ABB RobotStudio station: palletizing.rspag

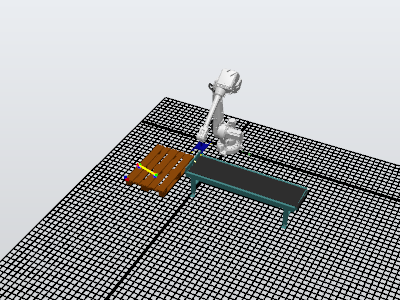
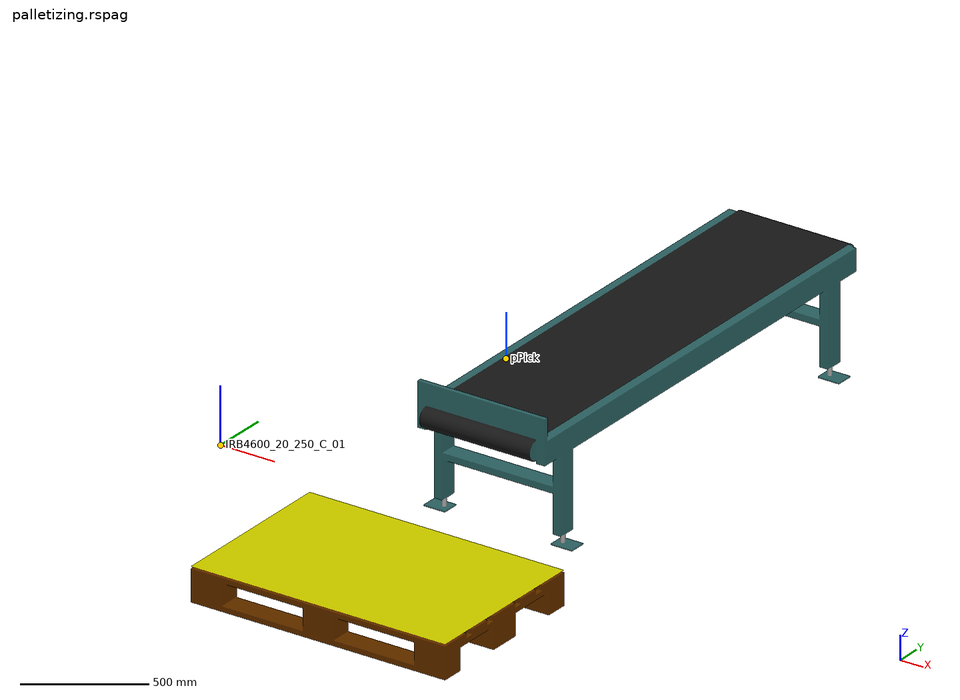
[picture v1: parts stored in the station drawn from their meshes, with robot base, taught points and paths (robot models come from the ABB library and are not in the file)]
--- station ---
Station palletizing (saved by RobotStudio 24.3.10958.1)
Controller IRB4600
  mechanical unit ROB_1: IRB4600_20_250_C_01, 6 joints, base frame (0, 0, 0) mm
Layout (positions relative to the parent item):
  - IRB4600_20_250_C_01 [mechanism, from %ABB.RobotStudio.Models.IRB4600%\IRB4600_20_250_C_G_01.rslib] at (0, 0, 0) mm; joint values [0.0538, -0.0275, 0.5427, 0, 1.0556, -1.517] (rad or m)
  - Belt Conveyor [part], size 703.5 x 2188.6 x 501 mm
  - Box [part], size 500 x 300 x 200 mm
  - SC_InFeeder [smart component]
      signals: DO doBoxInPos
      connections:
        LineSensor.SensorOut -> SC_InFeeder.doBoxInPos
        LineSensor.SensorOut -> LogicGate_2.InputA
        LogicGate_2.Output -> Source.Execute
    - Source [smart component, from Components\Source.rslib]
        properties: Source=Box; Copy=(none); Parent=(none); Position=[0 0 0]; Orientation=[0 0 0]; Transient=true; PhysicsBehavior=3
    - LineSensor [smart component, from Components\LineSensor.rslib]
        properties: Start=[1.3 -0.09 0.547]; End=[1.3 -0.03 0.547]; Radius=0; SensedPart=(none); SensedPoint=[1.3 -0.0800001220703125 0.547]; Length=0.06; Tag=(none)
      - _sensorPart_ [part], size 0 x 60 x 0 mm
    - LogicGate_2 [smart component, from Components\LogicGate.rslib]
        properties: Operator=NOT; Delay=0
  - Belt [part], size 529.1 x 2200.3 x 102.1 mm
  - Stop [part], size 600 x 20 x 100 mm
  - SC_VacuumTool [smart component] at (1300.02, 70, 1050.64) mm, rotated rx 180 ry 0 rz -90 deg
      signals: DI diAttach, DO doAttached
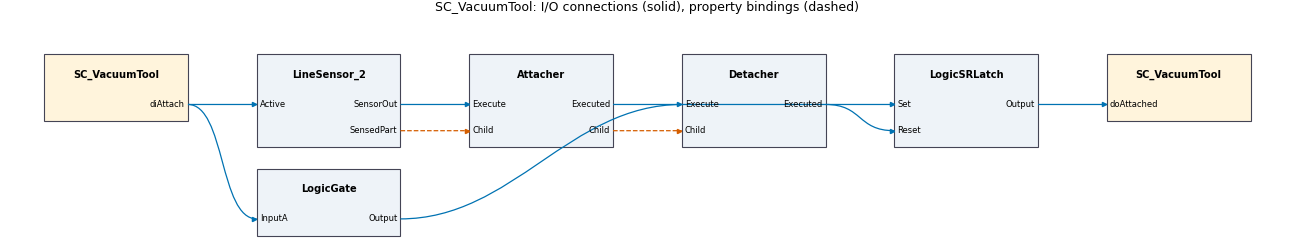
      connections:
        SC_VacuumTool.diAttach -> LineSensor_2.Active
        LineSensor_2.SensorOut -> Attacher.Execute
        Attacher.Executed -> LogicSRLatch.Set
        SC_VacuumTool.diAttach -> LogicGate.InputA
        LogicGate.Output -> Detacher.Execute
        Detacher.Executed -> LogicSRLatch.Reset
        LogicSRLatch.Output -> SC_VacuumTool.doAttached
        LineSensor_2.SensedPart => Attacher.Child
        Attacher.Child => Detacher.Child
    - LineSensor_2 [smart component, from Components\LineSensor.rslib]
        properties: Start=[0 0 0.1122]; End=[0 0 0.16]; Radius=0; SensedPart=(none); SensedPoint=[1.65000061035156 -1.05000048828125 0.345319213867188]; Length=0.0478; Tag=(none)
      - _sensorPart_ [part], size 0 x 0 x 47.8 mm
    - Attacher [smart component, from Components\Attacher.rslib]
        properties: Parent=Vacuum Tool; Flange=0; Child=(none); Mount=false; Offset=[0 0 0]; Orientation=[0 0 0]
    - Detacher [smart component, from Components\Detacher.rslib]
        properties: Child=(none); KeepPosition=true
    - LogicGate [smart component, from Components\LogicGate.rslib]
        properties: Operator=NOT; Delay=0
    - LogicSRLatch [smart component, from Components\LogicSRLatch.rslib]
    - Vacuum Tool [mechanism] at (0, 0, 0) mm
        TCP tVacuum at (0, 0, 150) mm
        links: Vacuum Tool
  - SC_OutFeeder [smart component]
      connections:
        PlaneSensor.SensorOut -> LogicGate.InputA
        LogicGate.Output -> Sink.Execute
        PlaneSensor.SensedPart => Sink.Object
    - EPAL Euro pallet [part] at (1900, -1200, 0) mm, rotated rx 0 ry 0 rz 90 deg, size 804.4 x 1206.6 x 151.6 mm
    - PlaneSensor [smart component, from Components\PlaneSensor.rslib]
        properties: Origin=[0.7 -1.2 0.154]; Axis1=[1.2 0 0]; Axis2=[0 0.8 0]; SensedPart=(none); Tag=(none)
      - _sensorPart_ [part], size 1200 x 800 x 0 mm
    - Sink [smart component, from Components\Sink.rslib]
        properties: Object=(none)
    - LogicGate [smart component, from Components\LogicGate.rslib]
        properties: Operator=NOP; Delay=2
Attachment: SC_VacuumTool is attached to IRB4600_20_250_C_01 / Link6
Station logic (signal -> signal, property => property):
  SC_VacuumTool.doAttached -> IRB4600.diVacuum
  IRB4600.doVacuum -> SC_VacuumTool.diAttach
  SC_InFeeder.doBoxInPos -> IRB4600.diBoxInPos
Targets, tools, work objects and paths stored in the station and not in the controller backup, written as RAPID:
! task T_ROB1
MODULE Module1
  PROC PickPart()
    MoveL pPick,v300,fine,tVacuum\WObj:=wobjInFeeder;
  ENDPROC
  PROC DropPart()
    MoveL Target_10,v300,fine,tVacuum\WObj:=wobjPallet;
    MoveL Target_20,v300,fine,tVacuum\WObj:=wobjPallet;
  ENDPROC
ENDMODULE


--- Backups/IRB4600/RAPID/TASK1/PROGMOD/CalibData.mod ---
MODULE CalibData
	PERS tooldata tVacuum:=[TRUE,[[0,0,150],[1,0,0,0]],[9,[0,0,100],[1,0,0,0],0,0,0]];
	TASK PERS wobjdata wobjInFeeder:=[FALSE,TRUE,"",[[0,0,0],[1,0,0,0]],[[1000,-80,497],[1,0,0,0]]];
    TASK PERS wobjdata wobjPallet:=[FALSE,TRUE,"",[[1900,-1200,144],[0.707106781,0,0,0.707106781]],[[0,0,0],[1,0,0,0]]];
ENDMODULE

--- Backups/IRB4600/RAPID/TASK1/PROGMOD/Module1.mod ---
MODULE Module1
    CONST robtarget pPick:=[[300.023,150,209.481],[0,-0.707106781,0.707106781,0],[0,0,0,0],[9E+09,9E+09,9E+09,9E+09,9E+09,9E+09]];
    CONST robtarget Target_10:=[[150,250,200],[0,0,1,0],[0,0,0,0],[9E+09,9E+09,9E+09,9E+09,9E+09,9E+09]];
    CONST robtarget Target_20:=[[550,150,200],[0,0.707106781,0.707106781,0],[-1,0,-1,0],[9E+09,9E+09,9E+09,9E+09,9E+09,9E+09]];
    !***********************************************************
    !
    ! Module:  Module1
    !
    ! Description:
    !   <Insert description here>
    !
    ! Author: ander
    !
    ! Version: 1.0
    !
    !***********************************************************


    !***********************************************************
    !
    ! Procedure main
    !
    !   Smart Component example, Pick and Place application.

    !
    !***********************************************************
    PROC main()
            Odd 0;
            Even 200;
            Odd 400;
            Even 600;
    ENDPROC

    PROC Odd(num offset)
        PickPart Offs(Target_10,0,0,offset);
        PickPart Offs(Target_10,0,700,offset);
        PickPart Offs(Target_20,0,0,offset);
        PickPart Offs(Target_20,0,300,offset);
        PickPart Offs(Target_20,0,600,offset);
        PickPart Offs(Target_20,0,900,offset);
    ENDPROC

    PROC Even(num offset)
        PickPart Offs(Target_10,500,0,offset);
        PickPart Offs(Target_10,500,700,offset);
        PickPart Offs(Target_20,-300,0,offset);
        PickPart Offs(Target_20,-300,300,offset);
        PickPart Offs(Target_20,-300,600,offset);
        PickPart Offs(Target_20,-300,900,offset);
    ENDPROC

    PROC PickPart(robtarget target)
        !** The robot moves to a wait position 200 mm above the pick position. **
        MoveJ Offs(pPick,0,0,200),v500,z1,tVacuum\WObj:=wobjInFeeder;
        !** The robot waits for a box to pick at the infeeder stop. **
        WaitDI diBoxInPos,1;
        !** The robot goes to the pick position. **
        MoveL pPick,v100,fine,tVacuum\WObj:=wobjInFeeder;
        !** To attach the box, the robot turns on the digital output signal "doVacuum" which is connected to the Smart Component "SC_VacuumTool". **
        SetDO doVacuum,1;
        !** The robot waits for the digital input signal "diVacuum" to goes high, which comes from "SC_VacuumTool" and indicates that the box is attached. **
        !WaitDI diVacuum,1;
        !** The robot moves up from the infeeder. **
        MoveL Offs(pPick,0,0,200),v500,z1,tVacuum\WObj:=wobjInFeeder;
        !** The robot moves to the drop position above the pallet. **
        DropPart target;
    ENDPROC

    PROC DropPart(robtarget target)
        VAR robtarget top_target;
        top_target:=Offs(target,0,0,400);

        MoveJ top_target,v500,z1,tVacuum\WObj:=wobjPallet;
        MoveL target,v100,fine,tVacuum\WObj:=wobjPallet;
        !** To detach the box, the robot turns off the digital output signal "doVacuum" which is connected to the Smart Component "SC_VacuumTool". **
        SetDO doVacuum,0;
        !** The robot waits for the digital input signal "diVacuum" to goes low, which comes from "SC_VacuumTool" and indicates that the box is detached. **
        !WaitDI diVacuum,0;
        !** The wait time simulates the time it takes for a real vacuum gripper to loose the vacuum. **
        WaitTime 0.5;
        MoveL top_target,v500,z1,tVacuum\WObj:=wobjPallet;
    ENDPROC
ENDMODULE

--- Backups/IRB4600/SYSPAR/EIO.cfg ---
EIO:CFG_1.0:6:1::
#
EIO_SIGNAL:

      -Name "doVacuum" -SignalType "DO" -Access "All"

      -Name "diVacuum" -SignalType "DI" -Access "All"

      -Name "diBoxInPos" -SignalType "DI" -Access "All"
